// TIA Portal V16 export
// export: Created 2022-04-14T22:35:56.5059968Z, ExportSetting WithDefaults, DisplayName Totally Integrated Automation Portal, DisplayVersion V16, DisplayName TIA Portal Version Control Interface, DisplayVersion V16, DisplayName TIA Portal Openness, DisplayVersion V16, DisplayName STEP 7 Professional, DisplayVersion V16, DisplayName STEP 7 Safety, DisplayVersion V16, DisplayName WinCC Professional, DisplayVersion V16
ORGANIZATION_BLOCK "Main"   // OB1, LAD, ProgramCycle
TITLE = "Main Program Sweep (Cycle)"
{ S7_Optimized_Access := 'TRUE' }
VERSION : 0.1
// stored: AutoNumber true, IsIECCheckEnabled false, SetENOAutomatically false
   VAR_INPUT
      Initial_Call : Bool;   // Initial call of this OB
      Remanence : Bool;   // =True, if remanent data are available
   END_VAR
BEGIN

REGION Network 1
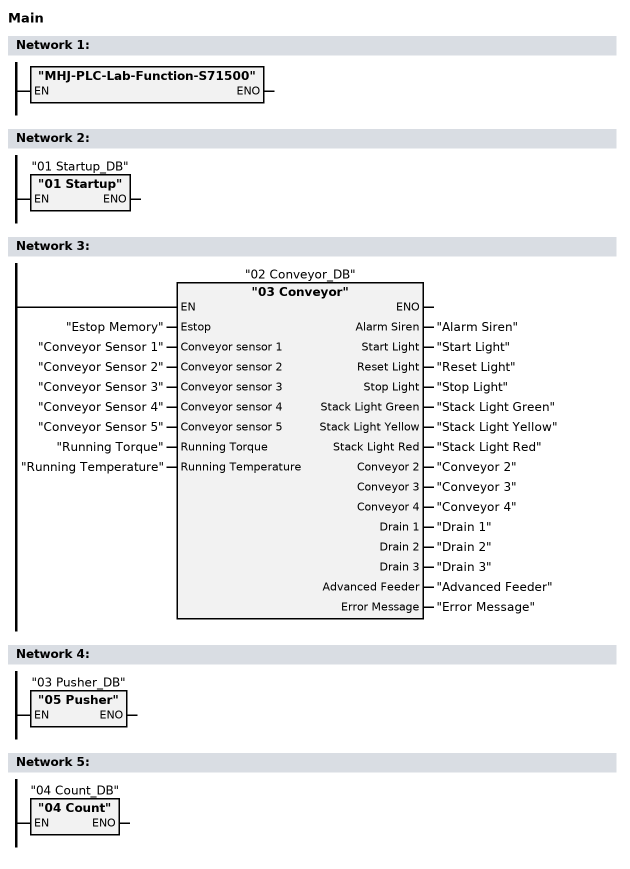
   RUNG wire#powerrail
      "MHJ-PLC-Lab-Function-S71500"()
   END_RUNG
   // the same network as SCL:
   "MHJ-PLC-Lab-Function-S71500"();
END_REGION

REGION Network 2
   RUNG wire#powerrail
      "01 Startup_DB"()
   END_RUNG
   // the same network as SCL:
   "01 Startup_DB"();   // "01 Startup"
END_REGION

REGION Network 3
   RUNG wire#powerrail
      "02 Conveyor_DB"(Estop := "Estop Memory", "Conveyor sensor 1" := "Conveyor Sensor 1", "Conveyor sensor 2" := "Conveyor Sensor 2", "Conveyor sensor 3" := "Conveyor Sensor 3", "Conveyor sensor 4" := "Conveyor Sensor 4", "Conveyor sensor 5" := "Conveyor Sensor 5", "Running Torque" := "Running Torque", "Running Temperature" := "Running Temperature", "Alarm Siren" => "Alarm Siren", "Start Light" => "Start Light", "Reset Light" => "Reset Light", "Stop Light" => "Stop Light", "Stack Light Green" => "Stack Light Green", "Stack Light Yellow" => "Stack Light Yellow", "Stack Light Red" => "Stack Light Red", "Conveyor 2" => "Conveyor 2", "Conveyor 3" => "Conveyor 3", "Conveyor 4" => "Conveyor 4", "Drain 1" => "Drain 1", "Drain 2" => "Drain 2", "Drain 3" => "Drain 3", "Advanced Feeder" => "Advanced Feeder", "Error Message" => "Error Message")
   END_RUNG
   // the same network as SCL:
   "02 Conveyor_DB"(Estop := "Estop Memory",   // "03 Conveyor"
                    "Conveyor sensor 1" := "Conveyor Sensor 1",
                    "Conveyor sensor 2" := "Conveyor Sensor 2",
                    "Conveyor sensor 3" := "Conveyor Sensor 3",
                    "Conveyor sensor 4" := "Conveyor Sensor 4",
                    "Conveyor sensor 5" := "Conveyor Sensor 5",
                    "Running Torque" := "Running Torque",
                    "Running Temperature" := "Running Temperature",
                    "Alarm Siren" => "Alarm Siren",
                    "Start Light" => "Start Light",
                    "Reset Light" => "Reset Light",
                    "Stop Light" => "Stop Light",
                    "Stack Light Green" => "Stack Light Green",
                    "Stack Light Yellow" => "Stack Light Yellow",
                    "Stack Light Red" => "Stack Light Red",
                    "Conveyor 2" => "Conveyor 2",
                    "Conveyor 3" => "Conveyor 3",
                    "Conveyor 4" => "Conveyor 4",
                    "Drain 1" => "Drain 1",
                    "Drain 2" => "Drain 2",
                    "Drain 3" => "Drain 3",
                    "Advanced Feeder" => "Advanced Feeder",
                    "Error Message" => "Error Message");
END_REGION

REGION Network 4
   RUNG wire#powerrail
      "03 Pusher_DB"()
   END_RUNG
   // the same network as SCL:
   "03 Pusher_DB"();   // "05 Pusher"
END_REGION

REGION Network 5
   RUNG wire#powerrail
      "04 Count_DB"()
   END_RUNG
   // the same network as SCL:
   "04 Count_DB"();   // "04 Count"
END_REGION
END_ORGANIZATION_BLOCK
